FUNCTION_BLOCK FB_NeutralFibreDetermine EXTENDS FB_Commons
(*************************************************************************************************)
(*  FILENAME:    FB_NeutralFibreDetermine                                                      *)
(*  PROJECT:     CALMAR PUPLC                                                                    *)
(*  COPYRIGHT:   All rights reserved (c) Wifag//Polytype, Fribourg/Switzerland (2022)            *)
(*  ENVIRONMENT: TwinCAT PLC                                                                     *)
(*  VERSION:     <version>                                                                       *)
(*************************************************************************************************)
(*  DESCRIPTION:                                                                   <description> *)
(*                                                                                </description> *)
(*************************************************************************************************)

{library public}
VAR_INPUT
  (*EL1252*)
  bIKp_MarkTrigger01        AT%I* : BOOL;        (*Mark sensor 01*)
  tIKp_TimeStampPos01       AT%I* : T_DCTIME64;  (*TimeStamp Pos_Edge @EL1252*)
  tIKn_TimeStampNeg01       AT%I* : T_DCTIME64;  (*TimeStamp Neg_Edge @EL1252*)
  bIKp_MarkTrigger02        AT%I* : BOOL;        (*Mark sensor 02*)
  tIKp_TimeStampPos02       AT%I* : T_DCTIME64;  (*TimeStamp Pos_Edge @EL1252*)
  tIKn_TimeStampNeg02       AT%I* : T_DCTIME64;  (*TimeStamp Neg_Edge @EL1252*)

  fI_ConveyorSpeed                : LREAL;       (*Current speed of substrate in [m/s]*)
END_VAR

VAR_OUTPUT
END_VAR

(*{library private}*)
VAR
  bInitOk                         : BOOL;           // initialized
  bSpeedValid                     : BOOL;           // speed is valid
  
  (*configuration*)
  _nResolution                    : INT := 1;       // Printhead Resolution [e.g. 600] x Subpixel Resolution [e.g. 32]*)

  fbRTrigMark01                   : R_TRIG;
  fbRTrigMark02                   : R_TRIG;
  
  fL_DurationMark01to02           : REAL;       (*Mark 1 to 2 [ms]*)
  fL_LengthMark01to02             : REAL;       (*Mark 1 to 2 [mm]*)
  nL_DeltaMark01to02              : DINT;       (*Mark 1 to 2 [SubPx]*)
END_VAR

IF NOT bInitOk THEN RETURN; END_IF;

fbRTrigMark01(CLK := bIKp_MarkTrigger01);
fbRTrigMark02(CLK := bIKp_MarkTrigger02);

IF fbRTrigMark01.Q THEN
	;
END_IF

IF fbRTrigMark02.Q THEN
	fL_DurationMark01to02 := LREAL_TO_REAL(ULINT_TO_LREAL(tIKp_TimeStampPos02) - ULINT_TO_LREAL(tIKp_TimeStampPos01)) / 1_000_000.0; (*[ms]*)
	fL_LengthMark01to02   := LREAL_TO_REAL((fL_DurationMark01to02 / 1000) * fI_ConveyorSpeed) * 1000;       (*[mm]*)
	nL_DeltaMark01to02    := LREAL_TO_DINT(fL_LengthMark01to02 * _nResolution / 25.4);  (*[SubPx]*)
END_IF

(********************************* END OF FB *****************************************************)

METHOD Init
VAR_INPUT
  nResolution                   : INT := 1;        (*Printhead Resolution [e.g. 600] x Subpixel Resolution [e.g. 32]*)
END_VAR
(*zero divisions*)
IF nResolution = 0 THEN 
  bInitOk := FALSE;

  RETURN; 
END_IF;

_nResolution := nResolution;

bInitOk := TRUE;
END_METHOD

END_FUNCTION_BLOCK

(* stored: Version 1.1.0.1, ProductVersion 3.1.4024.9
   POU FB_NeutralFibreDetermine: Id {09e5318c-d36f-4976-9501-8d59b352594a}, SpecialFunc None
   Method Init: Id {0e5d9d38-5568-4252-a7a4-4a674ac176b4} *)
